{attribute 'strict'}
TYPE E_CSVDataExchangerSelectAllState :
(
	CSV_DATA_EXCHANGER_SELECT_ALL_OPEN_FILE 			:= 0,
	CSV_DATA_EXCHANGER_SELECT_ALL_WAIT_FOR_OPENING		:= 10,	
	CSV_DATA_EXCHANGER_SELECT_ALL_READ_SINGLE_LINE 		:= 20,	
	CSV_DATA_EXCHANGER_SELECT_ALL_WAIT_FOR_READING		:= 30,	
	CSV_DATA_EXCHANGER_SELECT_ALL_PARSE_SINGLE_LINE		:= 40,	
	CSV_DATA_EXCHANGER_SELECT_ALL_CLOSE_FILE			:= 50,	
	CSV_DATA_EXCHANGER_SELECT_ALL_WAIT_FOR_CLOSING		:= 60,
	CSV_DATA_EXCHANGER_SELECT_ALL_READING_DONE			:= 70
);
END_TYPE

(* stored: Version 1.1.0.1, ProductVersion 3.1.4024.12
   DUT E_CSVDataExchangerSelectAllState: Id {fcae90b5-60c9-4689-b279-afb62b5db2c0} *)
